(* LS Electric XG5000 project: 05_Practice6_Counter_GT *)
(* PLC LSPLC *)
(* module base 0 slot 0: 입력 모듈:XGI-D21A (DC 24V 입력, 8점 (전류소스/싱크입력)) *)
(* module base 0 slot 1: 출력 모듈:XGQ-RY1A (릴레이 출력, 8점 (2A용, 단독 COM.)) *)

PROGRAM NewProgram (* task: 스캔 프로그램 *)
VAR
    PB0 AT %IX0.0.0 : BOOL;
    PB1 AT %IX0.0.1 : BOOL;
    리셋 : BOOL;
    모터1 AT %QX0.1.0 : BOOL;
    모터2 AT %QX0.1.1 : BOOL;
    모터3 AT %QX0.1.2 : BOOL;
    모터메모리1 AT %MX0 : BOOL;
    모터메모리2 AT %MX1 : BOOL;
    모터메모리3 AT %MX2 : BOOL;
    업카운터 : CTU_INT;
END_VAR

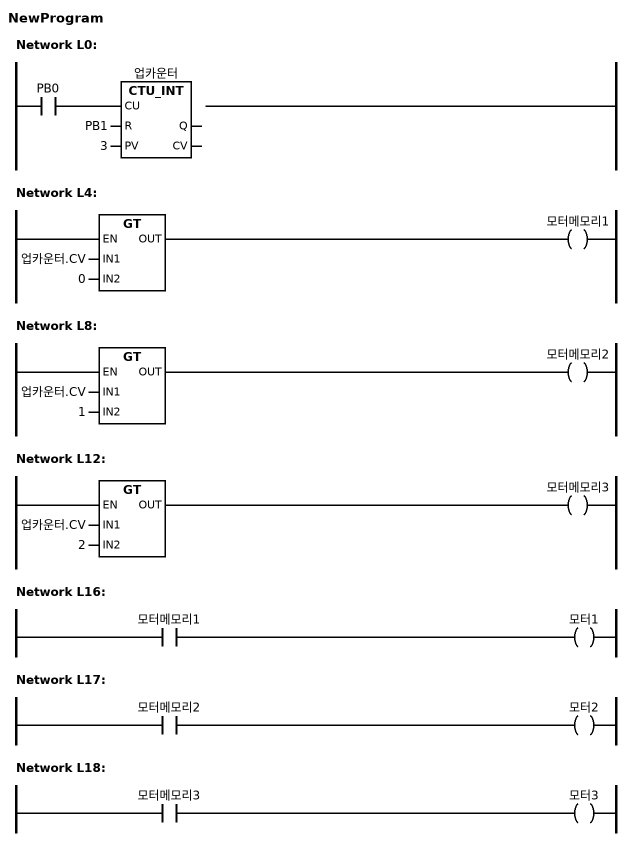
(* Rung L0 *)
업카운터(CU := PB0, R := PB1, PV := 3);
(* Rung L4 *)
모터메모리1 := 업카운터.CV > 0;
(* Rung L8 *)
모터메모리2 := 업카운터.CV > 1;
(* Rung L12 *)
모터메모리3 := 업카운터.CV > 2;
(* Rung L16 *)
모터1 := 모터메모리1;
(* Rung L17 *)
모터2 := 모터메모리2;
(* Rung L18 *)
모터3 := 모터메모리3;
END_PROGRAM